// TIA Portal V17 export
// export: Created 2024-09-15T12:29:53.9634087Z, ExportSetting WithDefaults, DisplayName Totally Integrated Automation Portal, DisplayVersion V17, DisplayName TIA Portal Openness, DisplayVersion V17, DisplayName TIA Portal Version Control Interface, DisplayVersion V17, DisplayName STEP 7 Professional, DisplayVersion V17, DisplayName STEP 7 Safety, DisplayVersion V17, DisplayName WinCC Professional, DisplayVersion V17
DATA_BLOCK "PRG_HBW_Axis_Vertical_Act_Pos_DB"   // DB28
AUTHOR : A.Schaefer
VERSION : 0.1
// stored: AutoNumber true, DBAccessibleFromOPCUA true, DBAccessibleFromWebserver true, InstanceOfName PRG_HBW_Axis_Vertical_Act_Pos, InstanceOfType FB
"PRG_HBW_Axis_Vertical_Act_Pos"
   // VAR
   //    lfb_IN_DEC { ExternalAccessible := 'False'; ExternalVisible := 'False'; ExternalWritable := 'False'} : "FB_INC_DEC";
   // END_VAR
BEGIN
END_DATA_BLOCK
